FUNCTION f_CalculateDeltaT : REAL

VAR_INPUT
	PowerInput : REAL ; // Watts
	Density : REAL ; // g/L
	SpecificHeatCapacity : REAL ; // j/(g C)
	Mass : REAL; // g
END_VAR

IF Density =0 OR SpecificHeatCapacity =0 OR Mass =0 THEN 
	f_CalculateDeltaT := 0 ; 
ELSIF Mass < 0.3 THEN  //Filter to prevent large spikes when dividing by very small mass numbers.
	f_CalculateDeltaT := 0 ; 
ELSE
	f_CalculateDeltaT := PowerInput / (Density * SpecificHeatCapacity * Mass);
END_IF

END_FUNCTION

(* stored: Version 1.1.0.1, ProductVersion 3.1.4024.12
   POU f_CalculateDeltaT: Id {67e8c0c9-d26a-4619-ac85-2e802df4f70d}, SpecialFunc None *)
